Fanuc KAREL source: KO00042.KL

PROGRAM KO00042
%NOLOCKGROUP
%ENVIRONMENT MIR
VAR
  P1: POSITION
  P2: XYZWPREXT
  F: BOOLEAN
  OUT: XYZWPR
BEGIN
  F = TRUE
  OUT = MIRROR(P1, P2, F)
END KO00042
